TYPE st_BMS_GetStatus :
STRUCT
	//Battery info
	BattInfo					:	st_MBMU_BatterySummary;
	
	//detailed info	
	MBMU_Status					:	st_MBMU_Status;
	SBMU						:	ARRAY[0..3] OF st_SBMU_Status;
	
	Events						:	st_BMS_Events;
END_STRUCT
END_TYPE

(* stored: Version 1.1.0.1, ProductVersion 3.1.4024.12
   DUT st_BMS_GetStatus: Id {005a8443-595a-4537-b6a8-503255910a5e} *)
